RoboDK station: cellSimulator-v7.rdk

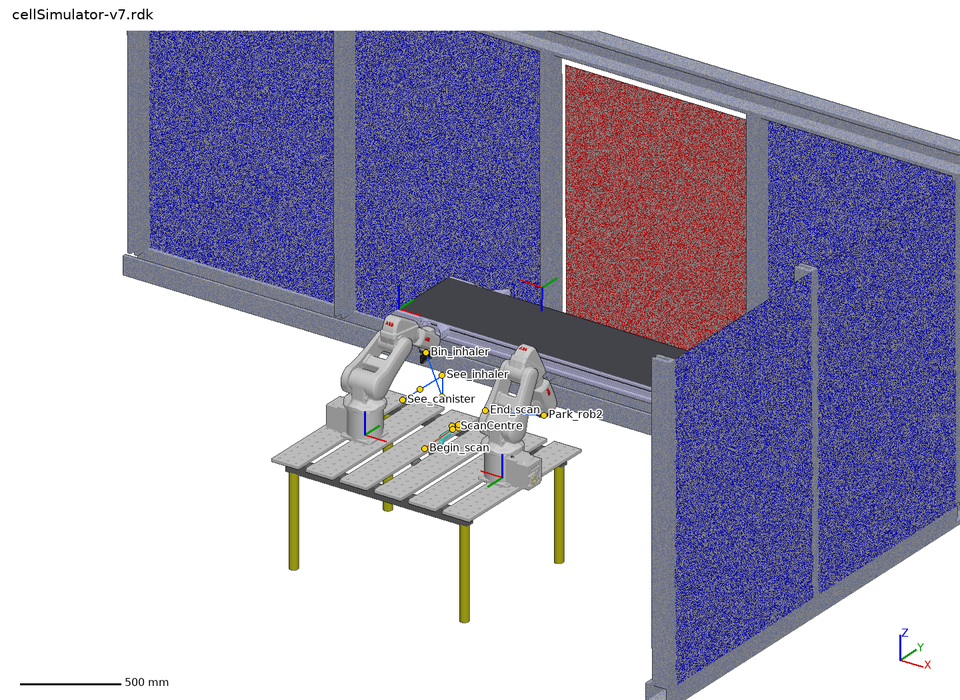
[picture v0: the station drawn from its stored meshes, robots at their saved joint values, targets as dots, program paths as lines]
Station ReMed_Demo_Sorting (saved by RoboDK 5.6.7). Poses are relative to the parent item; angles as X-Y-Z fixed-axis rotations.
  - object Table 1200x1000mm (Welding) at (30, 0, 0) mm, size 1193.8 x 965.2 x 609.6 mm, geometry from Table-1200x1000mm-Welding.sld
  - frame ABB IRB 120-3/0.6 Base at (-340, 0, 0) mm
    - robot ABB IRB 120-3/0.6: 6 axes, payload 3 kg, reach 580 mm, repeatability 0.01 mm, weight 25 kg
        modified DH rows (alpha deg, a mm, theta deg, d mm): 0, 0, 0, 290; -90, 0, -90, 0; 0, 270, 0, 0; -90, 70, 0, 302; 90, 0, 0, 0; -90, 0, 180, 72
        joint limits [-165, -110, -90, -160, -120, -400] to [165, 110, 70, 160, 120, 400]; home [0, 0, 0, 0, 0, 0]; saved at [90.543, 64.698, -33.139, 1.408, 58.437, 89.806]
      - robot Niryo Ned2 Gripper: 1 axes
          joint limits [0] to [43]; home [43]; saved at [43]
      - frame Niryo Ned2 Gripper Base at (-0.84, 1000, 39.99) mm
    - target See_canister (Cartesian target) at (340, -160, 350) mm, rotated rx 180 ry -1.2 rz 180 deg; joints [-25.104, 19.937, 16.254, -0.622, 54.897, -24.741] of ABB IRB 120-3/0.6
    - target See_canister2 (Cartesian target) at (340, -10.82, 350) mm, rotated rx 180 ry -1.2 rz 180 deg; joints [-1.816, 13.004, 25.062, -0.048, 53.134, -1.787] of ABB IRB 120-3/0.6
    - target See_inhaler (Cartesian target) at (340, 180, 350) mm, rotated rx -180 ry -1.2 rz 180 deg; joints [27.793, 21.681, 13.925, 0.679, 55.457, 27.402] of ABB IRB 120-3/0.6
    - target Pick_inhaler (Cartesian target) at (340, 180, 235) mm, rotated rx -180 ry -1.2 rz 180 deg; joints [27.793, 34.665, 19.804, 0.939, 36.596, 27.034] of ABB IRB 120-3/0.6
    - target Bin_inhaler (Cartesian target) at (-6.61, 538.04, 235) mm, rotated rx 180 ry -1.2 rz 180 deg; joints [90.543, 64.698, -33.139, 1.408, 58.437, 89.806] of ABB IRB 120-3/0.6
    - object Inhaler Main Assembly - Inhaler Body-1 at (366.28, 140, 34.92) mm, rotated rx 180 ry -1.2 rz 180 deg, size 28 x 84.9 x 50.6 mm, geometry from Inhaler Main Assembly - Inhaler Body-1.STL
    - object Constructed Body Canister STL - Inhaler Container 3-1 at (426.94, -160, 64.12) mm, rotated rx 180 ry -1.2 rz 180 deg, size 22 x 57.3 x 22 mm, geometry from Constructed Body Canister STL - Inhaler Container 3-1.STL
    - object Constructed Body Canister STL - Inhaler Container 3-1 at (426.94, -10, 64.12) mm, rotated rx 180 ry -1.2 rz 180 deg, size 22 x 57.3 x 22 mm, geometry from Constructed Body Canister STL - Inhaler Container 3-1.STL
  - program RobRight (10 instructions, listed below)
  - frame ABB IRB 120-3/0.6 Base at (493.01, -5.23, 0) mm, rotated rx 0 ry 0 rz -179.45 deg
    - robot ABB IRB 120-3/0.6: 6 axes, payload 3 kg, reach 580 mm, repeatability 0.01 mm, weight 25 kg
        modified DH rows (alpha deg, a mm, theta deg, d mm): 0, 0, 0, 290; -90, 0, -90, 0; 0, 270, 0, 0; -90, 70, 0, 302; 90, 0, 0, 0; -90, 0, 180, 72
        joint limits [-165, -110, -90, -160, -120, -400] to [165, 110, 70, 160, 120, 400]; home [0, 0, 0, 0, 0, 0]; saved at [-93.332, 29.188, 34.463, -4.669, 23.549, -88.295]
    - target Begin_scan (Cartesian target) at (291.74, 250.92, 180.78) mm, rotated rx -177.2 ry -1.98 rz 179.14 deg; joints [40.844, 43.342, 18.636, -1.486, 31.367, -317.057] of ABB IRB 120-3/0.6
    - target ScanCentre (Cartesian target) at (288.22, -14.32, 193.73) mm, rotated rx -177.2 ry -1.98 rz 179.14 deg; joints [-2.136, 27.968, 43.07, -7.925, 21.06, -353.879] of ABB IRB 120-3/0.6
    - target End_scan (Cartesian target) at (267.94, -240, 199.63) mm, rotated rx -177.2 ry -1.98 rz 179.14 deg; joints [-41.169, 36.097, 26.719, -7.51, 27.081, -393.676] of ABB IRB 120-3/0.6
    - target Park_rob2 (Cartesian target) at (-21.64, -331.35, 214.29) mm, rotated rx -177.22 ry -1.99 rz 179.15 deg; joints [-93.332, 29.188, 34.463, -4.669, 23.549, -88.295] of ABB IRB 120-3/0.6
    - target ScanUp (Cartesian target) at (311.5, -14.67, 192.93) mm, rotated rx -177.2 ry -1.98 rz 179.14 deg; joints [-2.041, 31.167, 37.627, -7.191, 23.289, 5.425] of ABB IRB 120-3/0.6
    - target ScanDown (Cartesian target) at (272.06, -14.08, 194.29) mm, rotated rx -177.2 ry -1.98 rz 179.14 deg; joints [-2.211, 25.752, 46.767, -8.505, 19.591, -353.337] of ABB IRB 120-3/0.6
    - target ScanLeft (Cartesian target) at (288.56, 11.61, 192.46) mm, rotated rx -177.2 ry -1.98 rz 179.14 deg; joints [2.967, 28.3, 42.923, -7.403, 21.098, -349.263] of ABB IRB 120-3/0.6
    - target ScanRight (Cartesian target) at (287.9, -38.46, 194.91) mm, rotated rx -177.2 ry -1.98 rz 179.14 deg; joints [-6.869, 27.929, 42.729, -8.282, 21.217, -358.29] of ABB IRB 120-3/0.6
  - program RobLeft_Ini (3 instructions, listed below)
  - program RobLeft_Scan1 (7 instructions, listed below)
  - program RobLeft_Scan2 (7 instructions, listed below)
  - program RobLeft_Scan3 (7 instructions, listed below)
  - program RobLeft_Scan4 (7 instructions, listed below)
  - program RobLeft_End (3 instructions, listed below)
  - program RobLeft (6 instructions, listed below)
  - object cage at (3037.5, 4079.46, -3012.56) mm, rotated rx 90 ry 0.21 rz -89.67 deg, size 2632.1 x 2052.6 x 5020 mm, geometry from cage.IGS
  - frame Conveyor Belt (2m) Base at (-1014.68, 1257.78, 0) mm
    - robot Conveyor Belt (2m): 1 axes
        modified DH rows (alpha deg, a mm, theta deg, d mm): 0, 0, 0, 0 linear
        base shift (0, 0, 0) mm, rotated rx 0 ry 90 rz 0 deg
        joint limits [-500000] to [500000]; home [0]; saved at [181.087]
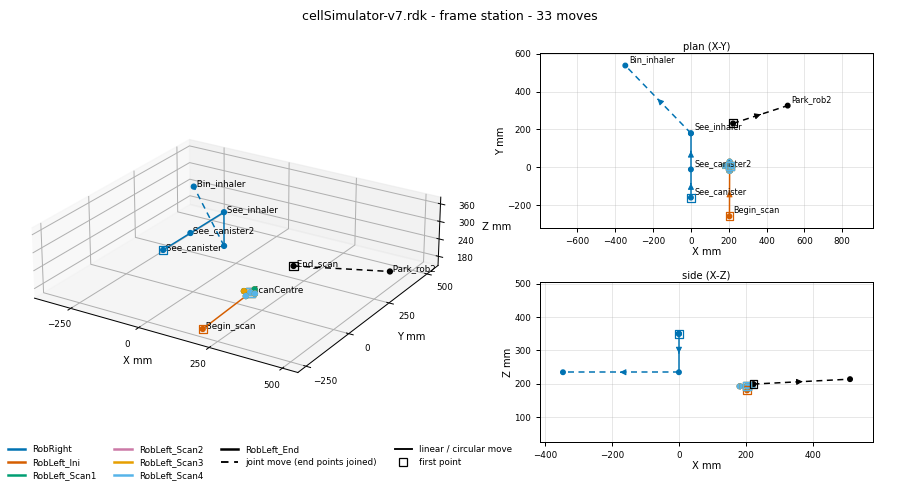
[picture p0: tool path of cellSimulator-v7.rdk in frame station, 33 of 33 moves have a stored position in this frame; points joined in program order, loops and branches not executed]

--- program RobRight (robot ABB IRB 120-3/0.6) ---
  Set Ref.: ABB IRB 120-3/0.6 Base
  MoveJ (See_canister)
  Pause 4.0 s
  MoveL (See_canister2)
  Pause 4.0 s
  MoveL (See_Inhaler) -> target See_inhaler
  Pause 4.0 s
  MoveL (Pick_Inhaler) -> target Pick_inhaler
  Pause 4.0 s
  MoveJ (Bin_Inhaler) -> target Bin_inhaler

--- program RobLeft_Ini (robot ABB IRB 120-3/0.6) ---
  Set Ref.: ABB IRB 120-3/0.6 Base
  MoveJ (Begin_scan)
  MoveL (ScanCentre)

--- program RobLeft_Scan1 (robot ABB IRB 120-3/0.6) ---
  Set Ref.: ABB IRB 120-3/0.6 Base
  MoveL (ScanCentre)
  MoveL (ScanUp)
  MoveL (ScanDown)
  MoveL (ScanCentre)
  MoveL (ScanLeft)
  MoveL (ScanRight)

--- program RobLeft_Scan2 (robot ABB IRB 120-3/0.6) ---
  Set Ref.: ABB IRB 120-3/0.6 Base
  MoveL (ScanCentre)
  MoveL (ScanUp)
  MoveL (ScanDown)
  MoveL (ScanCentre)
  MoveL (ScanLeft)
  MoveL (ScanRight)

--- program RobLeft_Scan3 (robot ABB IRB 120-3/0.6) ---
  Set Ref.: ABB IRB 120-3/0.6 Base
  MoveL (ScanCentre)
  MoveL (ScanUp)
  MoveL (ScanDown)
  MoveL (ScanCentre)
  MoveL (ScanLeft)
  MoveL (ScanRight)

--- program RobLeft_Scan4 (robot ABB IRB 120-3/0.6) ---
  Set Ref.: ABB IRB 120-3/0.6 Base
  MoveL (ScanCentre)
  MoveL (ScanUp)
  MoveL (ScanDown)
  MoveL (ScanCentre)
  MoveL (ScanLeft)
  MoveL (ScanRight)

--- program RobLeft_End (robot ABB IRB 120-3/0.6) ---
  Set Ref.: ABB IRB 120-3/0.6 Base
  MoveL (End_scan)
  MoveJ (Park_rob2)

--- program RobLeft (robot ABB IRB 120-3/0.6) ---
  Call RobLeft_Ini
  Call RobLeft_Scan1
  Call RobLeft_Scan2
  Call RobLeft_Scan3
  Call RobLeft_Scan4
  Call RobLeft_End
